FUNCTION SignalmappingOutput

(*=============== Digitale Ausgaenge ===============*)
GVL.mb_Input_Coils[3]	:=	Button_Start_LED;
GVL.mb_Input_Coils[4]	:=	Button_Stop_LED;
GVL.mb_Input_Coils[5]	:=	Button_Grundstellung_LED;
GVL.mb_Input_Coils[6]	:=	Button_Reset_LED;
GVL.mb_Input_Coils[7]	:=	Button_Quit_LED;
GVL.mb_Input_Coils[9]	:=	EmitterFeedIn;
GVL.mb_Input_Coils[10]	:=	FeedInForward;
GVL.mb_Input_Coils[11]	:=	FeedInStackerCraneForward;
GVL.mb_Input_Coils[12]	:=	RFIDFeedInExecuteCommand;
GVL.mb_Input_Coils[15]	:=	Gabel_zu_Pos_Links;
GVL.mb_Input_Coils[16]	:=	Gabel_zu_Pos_Rechts;
GVL.mb_Input_Coils[17]	:=	StackerCraneOneLiftFork;
GVL.mb_Input_Coils[19]	:=	ConveyorFeedOutStackerCrane;
GVL.mb_Input_Coils[20]	:=	ConveyorFeedOutTwoMeter;
GVL.mb_Input_Coils[21]	:=	ConveyorCurveFeedOut;
GVL.mb_Input_Coils[22]	:=	ConveyorFeedOutLong;
GVL.mb_Input_Coils[23]	:=	ConveyorFeedOutLongRemover;

(*=============== Analoge Ausgaenge ===============*)
GVL.mb_Input_Registers[3]	:=	RFIDFeedInCommand;
GVL.mb_Input_Registers[4]	:=	RFIDFeedInMemoryIndex;
GVL.mb_Input_Registers[5]	:=	RFIDFeedInWriteData;
GVL.mb_Input_Registers[7]	:=	StackerCraneOneTargetPos;

END_FUNCTION

(* stored: Version 1.1.0.1
   POU SignalmappingOutput: Id {2bdbb390-18c0-4372-a0ff-04e8c4b60455}, SpecialFunc None *)
